FUNCTION_BLOCK FT_DERIV_10_AR (* AR-Adapter-Wrapper um OSCAT FT_DERIV_10 - bruckt zwischen adapter und OSCAT, ohne dass eine der beiden Basisbibliotheken von der anderen abhaengt. K, Faktor und run als Klartext-InputVars durchgereicht (Default K=0, Faktor=1.0, run=TRUE) *)
  (* Standard: 61499-2; Description: Copyright (c) 2026 Meisterschulen am Ostbahnhof This program and the accompanying materials are made available under the terms of the Eclipse Public License 2.0 which is available at https://www.eclipse.org/legal/epl-2.0/ SPDX-License-Identifier: EPL-2.0 *)
  (* Version 1.1, 2026-09-20, Franz Höpfinger, Meisterschulen am Ostbahnhof, Bugfix: K/Faktor/run wurden nur per plain DataConnection an FT_DERIV_10 durchgereicht, ausgeloest einzig ueber AR_IN.E1 - kein Event auf diesem Wrapper hatte je eine With-Verknuepfung fuer diese Vars (IEC 61499 - ungebundene Vars werden nicht zuverlaessig gelesen). Neues explizites REQ-EventInput ergaenzt (parallel zu AR_IN.E1, beide -> FT_DERIV_10.REQ) mit With K/Faktor/run, gespiegelt vom inneren FT_DERIV_10.REQ. *)
  (* Version 1.0, 2026-09-12, Franz Höpfinger, Meisterschulen am Ostbahnhof, Initial implementation of FT_DERIV_10_AR wrapper FB *)
  PACKAGE OSCAT_adapter::Control;
  (* Documentation:
  FT_DERIV_10_AR
   🇩🇪 Deutsch
   AR-Adapter-Wrapper um OSCAT::Basic::POUs::Engineering::Control::FT_DERIV_10. K (Window Select, Default 0), Faktor (Multiplikationsfaktor, Default 1.0) und run (Berechnung aktiv, Default TRUE) sind Klartext-InputVars auf diesem Wrapper. Ein explizites REQ-EventInput (mit With K, With Faktor, With run) erlaubt den manuellen/periodischen Aufruf zusaetzlich zum automatischen Ausloesen ueber AR_IN.E1.
   Reine Adapter-Grenze
   Alle Hauptausgaenge von FT_DERIV_10 werden als eigene Adapter exponiert — kein Klartext-Event/-Datum verlaesst diesen Baustein:
    - AR_IN (Socket, AR): Eingangssignal (REAL, z. B. Impulszaehler-Rohwert von AD_TO_AR_NUM.AR_OUT)
   - AR_OUT (Plug, AR): die berechnete Ableitung (out, REAL, z. B. zur Weitergabe an CTRL_PID_AR.AR_ACT)
   - AUDI_DELTA_T (Plug, AUDI): Zeitdifferenz in Mikrosekunden (DT_0, UDINT)
   - AR_DELTA_IN (Plug, AR): Differenz des Eingangssignals (DI_0, REAL)
   - AB_VALID (Plug, AB): Gueltigkeit des Messpuffers (valid, BOOL)
    INIT/INITO und RST werden 1:1 an FT_DERIV_10.EINIT/.INITO/.RST durchgereicht.
   🇬🇧 English
   AR-adapter wrapper around OSCAT::Basic::POUs::Engineering::Control::FT_DERIV_10. K (window select, default 0), Faktor (multiplication factor, default 1.0) and run (calculation enabled, default TRUE) are plain InputVars on this wrapper. An explicit REQ event input (with With K, With Faktor, With run bindings) enables manual or periodic execution in addition to automatic triggering via AR_IN.E1.
   Pure Adapter Boundary
   All main outputs of FT_DERIV_10 are exposed as dedicated adapters:
    - AR_IN (Socket, AR): input signal (REAL)
   - AR_OUT (Plug, AR): calculated derivative (out, REAL)
   - AUDI_DELTA_T (Plug, AUDI): time difference in microseconds (DT_0, UDINT)
   - AR_DELTA_IN (Plug, AR): input signal difference (DI_0, REAL)
   - AB_VALID (Plug, AB): measurement buffer validity flag (valid, BOOL)
  *)
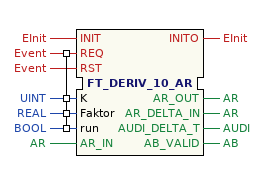
  EVENT_INPUT
    INIT : EInit; (* Service Initialization (durchgereicht an FT_DERIV_10.EINIT) *)
    REQ WITH K, Faktor, run; (* Explizite Ausfuehrungsanforderung (durchgereicht an FT_DERIV_10.REQ, zusaetzlich zu AR_IN.E1) *)
    RST; (* Reset der Ableitungshistorie (durchgereicht an FT_DERIV_10.RST) *)
  END_EVENT
  EVENT_OUTPUT
    INITO : EInit; (* Initialization Confirm *)
  END_EVENT
  VAR_INPUT
    K : UINT := 0; (* Window Select: 0=1 Period, 9=10 Periods (durchgereicht an FT_DERIV_10.K) *)
    Faktor : REAL := 1.0; (* Multiplikationsfaktor (durchgereicht an FT_DERIV_10.Faktor) *)
    run : BOOL := TRUE; (* Berechnung aktiv (durchgereicht an FT_DERIV_10.run) *)
  END_VAR
  SOCKETS
    AR_IN : adapter::types::unidirectional::AR; (* Eingangssignal (REAL) *)
  END_SOCKETS
  PLUGS
    AR_OUT : adapter::types::unidirectional::AR; (* Berechnete Ableitung (REAL, basierend auf K) *)
    AR_DELTA_IN : adapter::types::unidirectional::AR; (* Differenz des Eingangssignals ueber 1 Periode (REAL, DI_0) *)
    AUDI_DELTA_T : adapter::types::unidirectional::AUDI; (* Zeitdifferenz in Mikrosekunden ueber 1 Periode (UDINT, DT_0) *)
    AB_VALID : adapter::types::unidirectional::AB; (* Gueltigkeit der Messung (BOOL, durchgereicht von FT_DERIV_10.valid) *)
  END_PLUGS
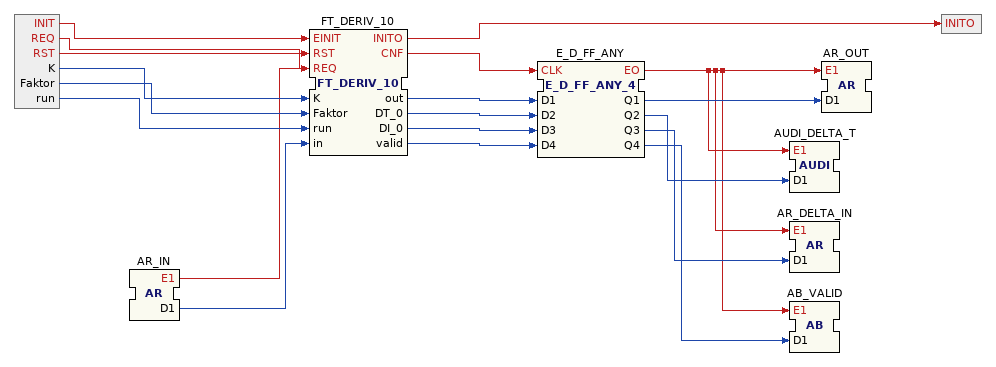
  FBS
    FT_DERIV_10 : OSCAT::Basic::POUs::Engineering::Control::FT_DERIV_10;
    E_D_FF_ANY : iec61499::events::E_D_FF_ANY_4;
  END_FBS
  EVENT_CONNECTIONS
    INIT TO FT_DERIV_10.EINIT;
    FT_DERIV_10.INITO TO INITO;
    RST TO FT_DERIV_10.RST;
    AR_IN.E1 TO FT_DERIV_10.REQ;
    REQ TO FT_DERIV_10.REQ;
    FT_DERIV_10.CNF TO E_D_FF_ANY.CLK;
    E_D_FF_ANY.EO TO AR_OUT.E1;
    E_D_FF_ANY.EO TO AUDI_DELTA_T.E1;
    E_D_FF_ANY.EO TO AR_DELTA_IN.E1;
    E_D_FF_ANY.EO TO AB_VALID.E1;
  END_CONNECTIONS
  DATA_CONNECTIONS
    K TO FT_DERIV_10.K;
    Faktor TO FT_DERIV_10.Faktor;
    run TO FT_DERIV_10.run;
    AR_IN.D1 TO FT_DERIV_10.in;
    FT_DERIV_10.out TO E_D_FF_ANY.D1;
    FT_DERIV_10.DT_0 TO E_D_FF_ANY.D2;
    FT_DERIV_10.DI_0 TO E_D_FF_ANY.D3;
    FT_DERIV_10.valid TO E_D_FF_ANY.D4;
    E_D_FF_ANY.Q1 TO AR_OUT.D1;
    E_D_FF_ANY.Q2 TO AUDI_DELTA_T.D1;
    E_D_FF_ANY.Q3 TO AR_DELTA_IN.D1;
    E_D_FF_ANY.Q4 TO AB_VALID.D1;
  END_CONNECTIONS
END_FUNCTION_BLOCK
